FUNCTION_BLOCK E_DEMUX_2 (* Service Interface Function Block Type *)
  (* Standard: 61499-2 *)
  (* Version 0.0, 2012-08-03, 4DIAC-IDE, 4DIAC-Consortium *)
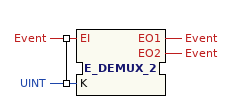
  EVENT_INPUT
    EI WITH K; (* execution request *)
  END_EVENT
  EVENT_OUTPUT
    EO1; (* Demux event output *)
    EO2; (* Demux event output *)
  END_EVENT
  VAR_INPUT
    K : UINT; (* Demux event number input *)
  END_VAR
  (* Service APPLICATION/RESOURCE: Service Interface Function Block Type *)
END_FUNCTION_BLOCK
